{attribute 'GeneratedUsingTerminal: EPP1322-0001-0017'}
{attribute addProperty BoxType "EPP1322-0001-0017"}
{attribute addProperty Id "A_0021_EPP1332_0001_0016A_0021_EPP1332_0001_0016_54E1D1AE378"}
{attribute addProperty CRC "3376102209"}
{attribute addProperty Size "378"}
TYPE A_0020_EPP1322_0001_0017_C93B3B41 EXTENDS EPP1322_1FC0878B :
STRUCT
	{attribute addProperty Name "A_0021(EPP1332-0001-0016)"}
	{attribute addProperty PreviousPort "A_0020(EPP1322-0001-0017) : D"}
	A_0021_EPP1332_0001_0016 : A_0021_EPP1332_0001_0016_54E1D1AE;
END_STRUCT
END_TYPE

(* stored: Version 1.2.0.0, ProductVersion 3.1.4024.9
   DUT A_0020_EPP1322_0001_0017_C93B3B41: Id {ec2cc31b-e99b-4c49-bdbd-52a8f0e53c6a} *)
